TYPE ST_PackMLBaseModule_HMI :
    STRUCT
        Config  : ST_PackMLBaseModule_Config;
        Command : ST_PackMLBaseModule_Command;
        Status  : ST_PackMLBaseModule_Status;
    END_STRUCT
END_TYPE

(* stored: Version 1.1.0.1, ProductVersion 3.1.4024.12
   DUT ST_PackMLBaseModule_HMI: Id {429b6452-115a-023b-26f1-81296929d633} *)
